Fanuc KAREL source: IO0224.KL

-- PROVISIONAL review KL for V770-1; original PC SHA256 ee433a754c2da05597d7d3f21cbf1aa92b7aae8ee3b9e5a5fc31193d5a2a2a87
-- Incomplete behavior may be omitted. Consult companion uncertainty JSON. Do not deploy.
PROGRAM IO0224
%NOLOCKGROUP
-- UNRESOLVED_LOCAL_POOL 5 cells at code offset 13; source declarations unknown
-- DIRECT_LOCAL_WORD_ACCESS alone does not prove INTEGER, REAL, or BOOLEAN
BEGIN
  -- UNRESOLVED_PC offsets 0-18; opcodes 2B,2C,7B
  -- UNRESOLVED_PC offsets 23-30; opcodes 9D,23
  -- UNRESOLVED_PC offsets 35-49; opcodes 2E,22,9D,33,35
  -- UNRESOLVED_PC offsets 54-61; opcodes 9D,23
  -- UNRESOLVED_PC offsets 66-77; opcodes 2E,23
  -- UNRESOLVED_PC offsets 82-132; opcodes 27,22,27,3F,27,3F,22,22,B0
  -- UNRESOLVED_PC offsets 137-141; opcodes 7F
  -- UNRESOLVED_PC offsets 146-150; opcodes 27,AA
  -- UNRESOLVED_PC offsets 155-159; opcodes 7F
END IO0224
